// Mitsubishi GX Works2 project: normal_servo_prj   PLC: Q03UDV

PROGRAM MAIN
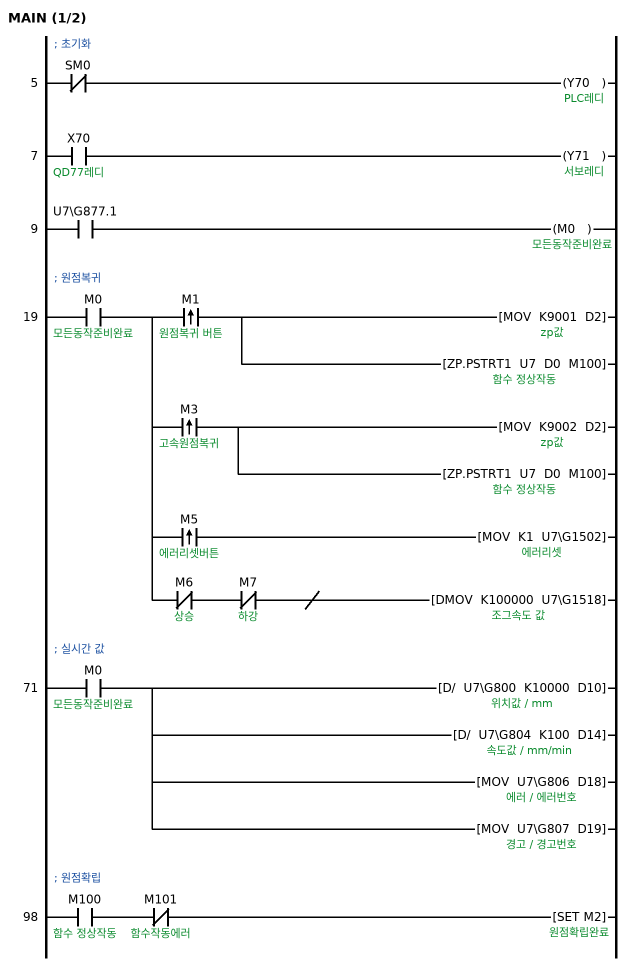
; 초기화
5     LDI     SM0
      OUT     Y70  ; PLC레디
7     LD      X70  ; QD77레디
      OUT     Y71  ; 서보레디
9     LD      U7\G877.1
      OUT     M0  ; 모든동작준비완료
; 원점복귀
19    LD      M0  ; 모든동작준비완료
      MPS
      ANDP    M1  ; 원점복귀 버튼
      MOV     K9001 D2  ; zp값
      ZP.PSTRT1 U7 D0 M100  ; 함수 정상작동
      MRD
      ANDP    M3  ; 고속원점복귀
      MOV     K9002 D2
      ZP.PSTRT1 U7 D0 M100
      MRD
      ANDP    M5  ; 에러리셋버튼
      MOV     K1 U7\G1502  ; 에러리셋
      MPP
      ANI     M6  ; 상승
      ANI     M7  ; 하강
      INV
      DMOV    K100000 U7\G1518  ; 조그속도 값
; 실시간 값
71    LD      M0  ; 모든동작준비완료
      D/      U7\G800 K10000 D10  ; 위치값 / mm
      D/      U7\G804 K100 D14  ; 속도값 / mm/min
      MOV     U7\G806 D18  ; 에러 / 에러번호
      MOV     U7\G807 D19  ; 경고 / 경고번호
; 원점확립
98    LD      M100  ; 함수 정상작동
      ANI     M101  ; 함수작동에러
      SET     M2  ; 원점확립완료
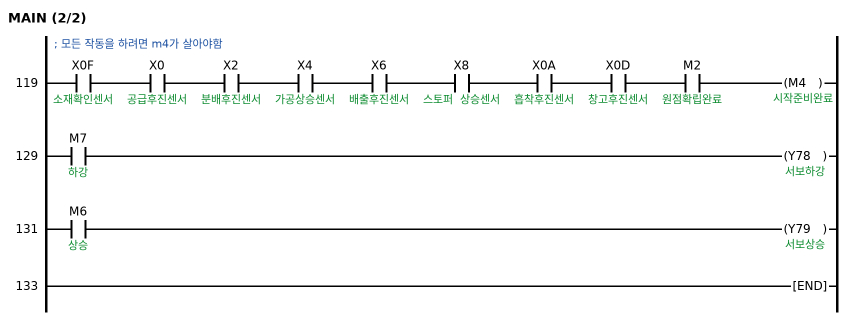
; 모든 작동을 하려면 m4가 살아야함
119   LD      X0F  ; 소재확인센서
      AND     X0  ; 공급후진센서
      AND     X2  ; 분배후진센서
      AND     X4  ; 가공상승센서
      AND     X6  ; 배출후진센서
      AND     X8  ; 스토퍼  상승센서
      AND     X0A  ; 흡착후진센서
      AND     X0D  ; 창고후진센서
      AND     M2  ; 원점확립완료
      OUT     M4  ; 시작준비완료
129   LD      M7  ; 하강
      OUT     Y78  ; 서보하강
131   LD      M6  ; 상승
      OUT     Y79  ; 서보상승
133   END
END_PROGRAM
